Fanuc KAREL source: main_task.kl

PROGRAM main_task
%NOBUSYLAMP
%COMMENT = ''
%NOLOCKGROUP
%NOPAUSESHFT
%NOPAUSE = COMMAND + TPENABLE + ERROR

-- [!IMPORTANT] THIS PROGRAM ONLY RUNS IN TEACH MODE. IT DOES NOT RUN IN AUTO

VAR
  motion_ctrl : INTEGER
  tsk_a_strt, tsk_b_strt : BOOLEAN
  tsk_a_done, tsk_b_done : BOOLEAN
  tmr : INTEGER
  status : INTEGER

%from display.klh %import clear, show
%include multitask.klh

BEGIN
  motion_ctrl = 1
  -- make motion control immediately available
  CLEAR_SEMA (motion_ctrl)
  POST_SEMA (motion_ctrl)

  display__clear
  WRITE TPDISPLAY(CR)
  WRITE TPDISPLAY(CR,'Running tasking example program.')
  WRITE TPDISPLAY(CR,'Press F1, or F2 to move robot')
  WRITE TPDISPLAY(CR,'Both tasks must be done before')
  WRITE TPDISPLAY(CR,'program exists.')
  display__show

  --start motions tasks
  tsk_a_strt = task__thread_motion('task_a', 1)
  tsk_b_strt = task__thread_motion('task_b', 1)

  REPEAT
    tsk_a_done = task__is_task_done('task_a')
    tsk_b_done = task__is_task_done('task_b')
    delay(100)
  UNTIL(tsk_a_done AND tsk_b_done)

  WRITE TPDISPLAY(CR,'program finished')

END main_task
